// TIA Portal V20 export
DATA_BLOCK "HMI_Interface_Parameter"   // DB262
// stored: Access Published, MemoryReserve 100
   VAR
      ProcessUnitSelect : Int := 5;   // 1. Anode Reel Cut, 2. Cathode Reel Cut, 3. Stacking#1, 4.Stacking#2, 5. Inspection
      Recipe : "HMI_IF_Parameter_LIstRecipe_Interface";
   END_VAR
   VAR RETAIN
      Parameter : Array[0..20] of "HMI_IF_Parameter_Parameter_UDT";
      Softcam : Array[0..23] of "LER_typeSoftCamRelation";
   END_VAR
   VAR
      RecipeButton : "HMI_IF_Parameter_Save Button_UDT";
      FATModeSelect : "LER_TypeFATMode_ModeSelect";
   END_VAR
   VAR RETAIN
      FATModeInterface : "LER_TypeFATModeInterface";
   END_VAR
   VAR
      teachingPosInterface { S7_SetPoint := 'True'} : Array[0..48] of "LER_TypeTeachingPosInterface";
      TeachingPos_Index { S7_SetPoint := 'True'} : SInt;
   END_VAR
BEGIN
END_DATA_BLOCK
